// Mitsubishi GX Works2 project: 타이머 무한반복   PLC: Q02/Q02H

PROGRAM MAIN
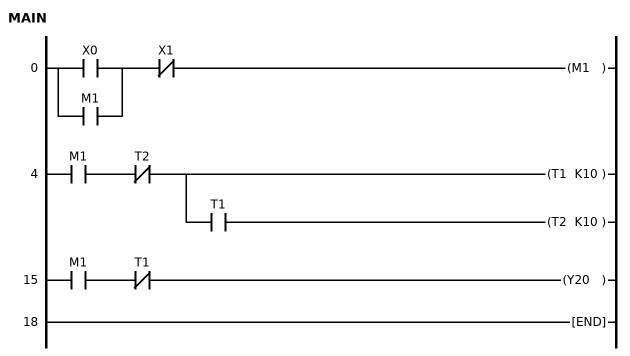
0     LD      X0
      OR      M1
      ANI     X1
      OUT     M1
4     LD      M1
      ANI     T2
      OUT     T1 K10
      AND     T1
      OUT     T2 K10
15    LD      M1
      ANI     T1
      OUT     Y20
18    END
END_PROGRAM
